PROGRAM SAFETY
VAR
END_VAR

IF SAFETY_IN.NOT_AUS_State=1 THEN

	FLAGS.SAFETY_OK:=TRUE;

ELSE

	FLAGS.SAFETY_OK:=FALSE;
END_IF;

END_PROGRAM

(* stored: Version 1.1.0.1, ProductVersion 3.1.0.26
   POU SAFETY: Id {43915553-f271-40f2-bf81-aae678947fef} *)
